(* PLC project Str_Capacity_TwinForge, TwinForge TwinForge 0.1.0 *)
(* stored: creationDateTime 2026-07-26T04:10:51.400129+00:00 *)

PROGRAM PLC_PRG
  VAR
    fbStrCapacity : Str_Capacity;
    xEnable : BOOL := TRUE;
    xEnableOut : BOOL;
    aData : ARRAY[0..9] OF SINT;
    diCapacity : DINT;
  END_VAR

                  fbStrCapacity(
    EnableIn := xEnable,
    EnableOut => xEnableOut,
    Ref_Data := aData,
    Val => diCapacity
);
                
END_PROGRAM

FUNCTION_BLOCK Str_Capacity
  VAR_INPUT
    EnableIn : BOOL;
  END_VAR
  VAR_OUTPUT
    EnableOut : BOOL;
    Val : DINT;
  END_VAR
  VAR_INPUT
    {attribute 'variable_length_array_original_scope' := 'Inout'}
    {attribute 'variable_length_array' := 'ARRAY[*] OF SINT'}
    {attribute 'Dimensions' := '1'}
    Ref_Data : POINTER TO SINT;
  END_VAR

                  EnableOut := EnableIn;
IF EnableIn THEN
    Val := ((UPPER_BOUND(Ref_Data, (0 + 1)) - LOWER_BOUND(Ref_Data, (0 + 1))) + 1);
END_IF;
                
END_FUNCTION_BLOCK

CONFIGURATION Application
  RESOURCE Application ON PLC
    TASK MainTask(INTERVAL := T#20ms, PRIORITY := 1);
    PROGRAM PLC_PRG WITH MainTask : PLC_PRG;
  END_RESOURCE
END_CONFIGURATION
